	A	XV008_OPN 	// XV008.QOPEN = true
	JCN L67

	L   840
	T   stepnumber

L67: NOP 0


D67: NOP 0	

//---------------------------------
// End of network: jump here if step not active
// Jump to end of this FB if the step has been active to avoid
// execution of another step in the same scan
//---------------------------------		
	JU	ENDS
J67: NOP 0

NETWORK
TITLE = Step 840
// test dot-format to Linked CM in assignment => should convert to suffix
// skip this network if stepnumber not equal to 840
	L 	stepnumber
	L 	840
	==I
	JCN J68

//---------------------------------
// Actions (continuouss)
//---------------------------------

// Action: XV003.AUT_OP = true
	SET
	=	XV003_CMD

//---------------------------------
// --- TRANSITION TO S850 ---
//---------------------------------

// Transition Logic
	SET	// make sure RLO is high so the transition can happen when no conditions present

	JCN L68

	L   850
	T   stepnumber

L68: NOP 0


D68: NOP 0	

//---------------------------------
// End of network: jump here if step not active
// Jump to end of this FB if the step has been active to avoid
// execution of another step in the same scan
//---------------------------------		
	JU	ENDS
J68: NOP 0

NETWORK
TITLE = Step 850
// test dot-format from Linked CM in evaluation =>should convert to suffix
// skip this network if stepnumber not equal to 850
	L 	stepnumber
	L 	850
	==I
	JCN J69

//---------------------------------
// Actions (continuouss)
//---------------------------------

//---------------------------------
// --- TRANSITION TO S860 ---
//---------------------------------

// Transition Logic
	SET	// make sure RLO is high so the transition can happen when no conditions present

	A	XV003_OPN 	// XV003.QOPEN = true
	JCN L69

	L   860
	T   stepnumber

L69: NOP 0


D69: NOP 0	

//---------------------------------
// End of network: jump here if step not active
// Jump to end of this FB if the step has been active to avoid
// execution of another step in the same scan
//---------------------------------		
	JU	ENDS
J69: NOP 0

NETWORK
TITLE = Step 860
// test direct access to an EM instance in dot-format in the assignment => should stay in dot-format
// skip this network if stepnumber not equal to 860
	L 	stepnumber
	L 	860
	==I
	JCN J70

//---------------------------------
// Actions (continuouss)
//---------------------------------

// Action: EM_Instance_4.Pressure_SP  = 4.2
	L 	4.2
	T 	cstate.Equipment_Modules.EM_Instance_4.Pressure_SP

//---------------------------------
// --- TRANSITION TO S870 ---
//---------------------------------

// Transition Logic
	SET	// make sure RLO is high so the transition can happen when no conditions present

	JCN L70

	L   870
	T   stepnumber

L70: NOP 0


D70: NOP 0	

//---------------------------------
// End of network: jump here if step not active
// Jump to end of this FB if the step has been active to avoid
// execution of another step in the same scan
//---------------------------------		
	JU	ENDS
J70: NOP 0

NETWORK
TITLE = Step 870
// test direct access to a EM in dot-notation in the evaluation => should stay in dot-format
// skip this network if stepnumber not equal to 870
	L 	stepnumber
	L 	870
	==I
	JCN J71

//---------------------------------
// Actions (continuouss)
//---------------------------------

//---------------------------------
// --- TRANSITION TO S880 ---
//---------------------------------

// Calculation: cstate.Equipment_Modules.EM_Instance_4.Level >= 50.0
	L 	cstate.Equipment_Modules.EM_Instance_4.Level
	L 	50.0
	>=R
	=	B12

// Transition Logic
	SET	// make sure RLO is high so the transition can happen when no conditions present

	A	B12 	// EM_Instance_4.Level >= 50.0
	JCN L71

	L   880
	T   stepnumber

L71: NOP 0


D71: NOP 0	

//---------------------------------
// End of network: jump here if step not active
// Jump to end of this FB if the step has been active to avoid
// execution of another step in the same scan
//---------------------------------		
	JU	ENDS
J71: NOP 0

NETWORK
TITLE = Step 880
// test dot-format to Linked EM in assignment => should stay in dot-format
// skip this network if stepnumber not equal to 880
	L 	stepnumber
	L 	880
	==I
	JCN J72

//---------------------------------
// Actions (continuouss)
//---------------------------------

// Action: Some_Dyn_EM.Pressure_SP  = 4.2
	L 	4.2
	T 	Some_Dyn_EM.Pressure_SP

//---------------------------------
// --- TRANSITION TO S890 ---
//---------------------------------

// Transition Logic
	SET	// make sure RLO is high so the transition can happen when no conditions present

	JCN L72

	L   890
	T   stepnumber

L72: NOP 0


D72: NOP 0	

//---------------------------------
// End of network: jump here if step not active
// Jump to end of this FB if the step has been active to avoid
// execution of another step in the same scan
//---------------------------------		
	JU	ENDS
J72: NOP 0

NETWORK
TITLE = Step 890
// test dot-format from Linked EM in evaluation =>should stay in dot-format
// skip this network if stepnumber not equal to 890
	L 	stepnumber
	L 	890
	==I
	JCN J73

//---------------------------------
// Actions (continuouss)
//---------------------------------

//---------------------------------
// --- TRANSITION TO S910 ---
//---------------------------------

// Calculation: Some_Dyn_EM.Level >= 50.0
	L 	Some_Dyn_EM.Level
	L 	50.0
	>=R
	=	B13

// Transition Logic
	SET	// make sure RLO is high so the transition can happen when no conditions present

	A	B13 	// Some_Dyn_EM.Level >= 50.0
	JCN L73

	L   910
	T   stepnumber

L73: NOP 0


D73: NOP 0	

//---------------------------------
// End of network: jump here if step not active
// Jump to end of this FB if the step has been active to avoid
// execution of another step in the same scan
//---------------------------------		
	JU	ENDS
J73: NOP 0

NETWORK
TITLE = Step 910
// test suffix-format to Linked EM in assignment => should convert to dot-format
// skip this network if stepnumber not equal to 910
	L 	stepnumber
	L 	910
	==I
	JCN J74

//---------------------------------
// Actions (continuouss)
//---------------------------------

// Action: Some_Dyn_EM_P_SP  = 4.3
	L 	4.3
	T 	Some_Dyn_EM.Pressure_SP

//---------------------------------
// --- TRANSITION TO S920 ---
//---------------------------------

// Transition Logic
	SET	// make sure RLO is high so the transition can happen when no conditions present

	JCN L74

	L   920
	T   stepnumber

L74: NOP 0


D74: NOP 0	

//---------------------------------
// End of network: jump here if step not active
// Jump to end of this FB if the step has been active to avoid
// execution of another step in the same scan
//---------------------------------		
	JU	ENDS
J74: NOP 0

NETWORK
TITLE = Step 920
// test suffix-format from Linked EM in evaluation =>should convert to dot-format
// skip this network if stepnumber not equal to 920
	L 	stepnumber
	L 	920
	==I
	JCN J75

//---------------------------------
// Actions (continuouss)
//---------------------------------

//---------------------------------
// --- TRANSITION TO S930 ---
//---------------------------------

// Calculation: Some_Dyn_EM.Level >= 50.0
	L 	Some_Dyn_EM.Level
	L 	50.0
	>=R
	=	B14

// Transition Logic
	SET	// make sure RLO is high so the transition can happen when no conditions present

	A	B14 	// Some_Dyn_EM_LT  >= 50.0
	JCN L75

	L   930
	T   stepnumber

L75: NOP 0


D75: NOP 0	

//---------------------------------
// End of network: jump here if step not active
// Jump to end of this FB if the step has been active to avoid
// execution of another step in the same scan
//---------------------------------		
	JU	ENDS
J75: NOP 0

NETWORK
TITLE = Step 930
// write a bool
// skip this network if stepnumber not equal to 930
	L 	stepnumber
	L 	930
	==I
	JCN J76

//---------------------------------
// Actions (continuouss)
//---------------------------------

// Action: some_bool_out = true
	SET
	=	some_bool_out

//---------------------------------
// --- TRANSITION TO S940 ---
//---------------------------------

// Transition Logic
	SET	// make sure RLO is high so the transition can happen when no conditions present

	JCN L76

	L   940
	T   stepnumber

L76: NOP 0


D76: NOP 0	

//---------------------------------
// End of network: jump here if step not active
// Jump to end of this FB if the step has been active to avoid
// execution of another step in the same scan
//---------------------------------		
	JU	ENDS
J76: NOP 0

NETWORK
TITLE = Step 940
// test absolute value calculation
// skip this network if stepnumber not equal to 940
	L 	stepnumber
	L 	940
	==I
	JCN J77

//---------------------------------
// Actions (continuouss)
//---------------------------------

// Action: test1 = abs(2.3)
	L	2.3
	ABS
	T	test1

// Action: test2 = abs(test1)
	L	test1
	ABS
	T	test2

//---------------------------------
// --- TRANSITION TO S950 ---
//---------------------------------

// Transition Logic
	SET	// make sure RLO is high so the transition can happen when no conditions present

	JCN L77

	L   950
	T   stepnumber

L77: NOP 0


D77: NOP 0	

//---------------------------------
// End of network: jump here if step not active
// Jump to end of this FB if the step has been active to avoid
// execution of another step in the same scan
//---------------------------------		
	JU	ENDS
J77: NOP 0

NETWORK
TITLE = Step 950
// test absolute value calculation to int value
// skip this network if stepnumber not equal to 950
	L 	stepnumber
	L 	950
	==I
	JCN J78

//---------------------------------
// Actions (continuouss)
//---------------------------------

// Action: intvar = abs(4.6)
	L	4.6
	ABS
	RND;
	T	intvar

// Action: intvar = abs(test1)
	L	test1
	ABS
	RND;
	T	intvar

// Calculation: abs(3.2)
	L 	3.2
	ABS
	T 	V16

// Calculation: intvar + (abs(3.2))
	L 	intvar
	ITD;
DTR;
	L 	V16
	+R
	T 	V17

// Action: intvar = intvar + (intvar+ abs(3.2))
	L	intvar
	ITD;
DTR;
	L	V17
	+I
	RND;
	T	intvar

//---------------------------------
// --- TRANSITION TO S960 ---
//---------------------------------

// Transition Logic
	SET	// make sure RLO is high so the transition can happen when no conditions present

	JCN L78

	L   960
	T   stepnumber

L78: NOP 0


D78: NOP 0	

//---------------------------------
// End of network: jump here if step not active
// Jump to end of this FB if the step has been active to avoid
// execution of another step in the same scan
//---------------------------------		
	JU	ENDS
J78: NOP 0

NETWORK
TITLE = Step 960
// test absolut function of another calc
// skip this network if stepnumber not equal to 960
	L 	stepnumber
	L 	960
	==I
	JCN J79

//---------------------------------
// Actions (continuouss)
//---------------------------------

// Calculation: test1 + test2
	L 	test1
	L 	test2
	+R
	T 	V18

// Action: test1 = abs(test1 + test2)
	L	V18
	ABS
	T	test1

//---------------------------------
// --- TRANSITION TO S970 ---
//---------------------------------

// Transition Logic
	SET	// make sure RLO is high so the transition can happen when no conditions present

	JCN L79

	L   970
	T   stepnumber

L79: NOP 0


D79: NOP 0	

//---------------------------------
// End of network: jump here if step not active
// Jump to end of this FB if the step has been active to avoid
// execution of another step in the same scan
//---------------------------------		
	JU	ENDS
J79: NOP 0

NETWORK
TITLE = Step 970
// test multiple transitions in one step
// skip this network if stepnumber not equal to 970
	L 	stepnumber
	L 	970
	==I
	JCN J80

//---------------------------------
// Actions (continuouss)
//---------------------------------

//---------------------------------
// --- TRANSITION TO S980 ---
//---------------------------------

// Calculation: foo > 1.0
	L 	foo
	L 	1.0
	>R
	=	B15

// Transition Logic
	SET	// make sure RLO is high so the transition can happen when no conditions present

	A	B15 	// foo > 1.0
	JCN L80

	L   980
	T   stepnumber

L80: NOP 0

//---------------------------------
// --- TRANSITION TO S990 ---
//---------------------------------

// Calculation: foo <= 1.0
	L 	foo
	L 	1.0
	<=R
	=	B16

// Transition Logic
	SET	// make sure RLO is high so the transition can happen when no conditions present

	A	B16 	// foo <= 1.0
	JCN L81

	L   990
	T   stepnumber

L81: NOP 0


D80: NOP 0	

//---------------------------------
// End of network: jump here if step not active
// Jump to end of this FB if the step has been active to avoid
// execution of another step in the same scan
//---------------------------------		
	JU	ENDS
J80: NOP 0

NETWORK
TITLE = Step 980
// assignment where the right part is a boolean variable
// skip this network if stepnumber not equal to 980
	L 	stepnumber
	L 	980
	==I
	JCN J81

//---------------------------------
// Actions (continuouss)
//---------------------------------

// Action: Bool1 = Bool2
	A	Bool2
	=	Bool1

//---------------------------------
// --- TRANSITION TO S990 ---
//---------------------------------

// Transition Logic
	SET	// make sure RLO is high so the transition can happen when no conditions present

	JCN L82

	L   990
	T   stepnumber

L82: NOP 0


D81: NOP 0	

//---------------------------------
// End of network: jump here if step not active
// Jump to end of this FB if the step has been active to avoid
// execution of another step in the same scan
//---------------------------------		
	JU	ENDS
J81: NOP 0

NETWORK
TITLE = Step 990
// comparison where the right part is a boolen variable
// skip this network if stepnumber not equal to 990
	L 	stepnumber
	L 	990
	==I
	JCN J82

//---------------------------------
// Actions (continuouss)
//---------------------------------

//---------------------------------
// --- TRANSITION TO S1000 ---
//---------------------------------

// Calculation: Bool1 == Bool2
	X 	Bool1
	X 	Bool2
	NOT
	=	B17	// use of XOR to compare two bools

// Transition Logic
	SET	// make sure RLO is high so the transition can happen when no conditions present

	A	B17 	// Bool1 = Bool2
	JCN L83

	L   1000
	T   stepnumber

L83: NOP 0


D82: NOP 0	

//---------------------------------
// End of network: jump here if step not active
// Jump to end of this FB if the step has been active to avoid
// execution of another step in the same scan
//---------------------------------		
	JU	ENDS
J82: NOP 0

NETWORK
TITLE = Step 1000
// function call
// skip this network if stepnumber not equal to 1000
	L 	stepnumber
	L 	1000
	==I
	JCN J83

//---------------------------------
// Actions (continuouss)
//---------------------------------

// Action: function call: write_to_DB_DW (50, 20, 123)
	CALL write_to_DB_DW
	DB_NO := 50
	Location := 20
	Value := 123

// Action: function call: write_to_DB_DW (DB_NO, 20, 123)
	CALL write_to_DB_DW
	DB_NO := DB_NO
	Location := 20
	Value := 123

// Action: function call: intvar = somefunction(34,32)
	CALL somefunction
	arg1 := 34
	arg2 := 32

//---------------------------------
// --- TRANSITION TO S0 ---
//---------------------------------

// Transition Logic
	SET	// make sure RLO is high so the transition can happen when no conditions present

	JCN L84

	L   0
	T   stepnumber

L84: NOP 0


D83: NOP 0	

//---------------------------------
// End of network: jump here if step not active
// Jump to end of this FB if the step has been active to avoid
// execution of another step in the same scan
//---------------------------------		
	JU	ENDS
J83: NOP 0

NETWORK
TITLE = Step 8000
// Holding
// skip this network if stepnumber not equal to 8000
	L 	stepnumber
	L 	8000
	==I
	JCN J84

//---------------------------------
// Actions (continuouss)
//---------------------------------

//---------------------------------
// --- TRANSITION TO S8990 ---
//---------------------------------

// Transition Logic
	SET	// make sure RLO is high so the transition can happen when no conditions present

	JCN L85

	L   8990
	T   stepnumber

L85: NOP 0


D84: NOP 0	

//---------------------------------
// End of network: jump here if step not active
// Jump to end of this FB if the step has been active to avoid
// execution of another step in the same scan
//---------------------------------		
	JU	ENDS
J84: NOP 0

NETWORK
TITLE = END OF THE STEPS AND TRANSITIONS
// ################################
// ################################
// Placeholder network to indicate the end of the actual sequence
// ################################	  
// ################################
// jump location for the step that is currently active
ENDS:	NOP 0

NETWORK
TITLE = Write EMs
// network comment

	CALL em_write 
	   EM_ID                    := EM_I_OUT_ID
	   UDT_LOCATION             := #EM_I_OUT
	   UDT_OFFSET               := 40
	   Length                   := 40
	   Request					:=EM_I_OUT.Request
	   Owner					:=EM_I_OUT.Owner
	   EM_addressing_error      := M      0.0
	   RETVAL                   := MW     0

	CALL em_write 
	   EM_ID                    := Some_Dyn_EM_ID
	   UDT_LOCATION             := #Some_Dyn_EM
	   UDT_OFFSET               := 40
	   Length                   := 40
	   Request					:=Some_Dyn_EM.Request
	   Owner					:=Some_Dyn_EM.Owner
	   EM_addressing_error      := M      0.0
	   RETVAL                   := MW     0

NETWORK
TITLE = title
// network comment
// empty placeholder network
END_FUNCTION_BLOCK
